{attribute 'GeneratedUsingTerminal: EL7201-0000-0017'}
{attribute addProperty BoxType "EL7201-0000-0017"}
{attribute addProperty Id "Target_velocityAT %Q*DINT4"}
{attribute addProperty CRC "145315899"}
{attribute addProperty Size "4"}
TYPE DRV_Target_velocity_08A9583B :
STRUCT
	{attribute addProperty Name "Target_velocity"}
	Target_velocity AT %Q* : DINT;
END_STRUCT
END_TYPE

(* stored: Version 1.2.0.0, ProductVersion 3.1.4024.9
   DUT DRV_Target_velocity_08A9583B: Id {0ef27f52-cc66-4ce2-ab73-5e86e4e843b0} *)
